(* PLC project liner_cyclic.project, CODESYS CODESYS V3.5 SP17 Patch 3 *)
(* stored: creationDateTime 1970-01-01T00:00:00, modificationDateTime 1970-01-01T00:00:00 *)

PROGRAM SafetyChain
  VAR
    BLINK_0 : BLINK;
    bHomePosition : BOOL;
    R_TRIG_0 : R_TRIG;
    UP : BOOL;
    DOWN : BOOL;
    R_TRIG_2 : R_TRIG;
    tTimeLow : TIME := TIME#1s0ms;
    tTimeHigh : TIME := TIME#2s0ms;
    GREEN : BOOL;
    BLINK_1 : BLINK;
    GREEN_BLINK : BOOL;
    out_blink : BOOL;
    R_TRIG_8 : R_TRIG;
    TON_0 : TON;
    R_TRIG_1 : R_TRIG;
    RED : BOOL;
  END_VAR
  VAR  (* added by the conversion: wires and edge detectors of the diagram *)
    _GE47_ENO : BOOL;
    _GE47_OUT : BOOL;
    _LE51_ENO : BOOL;
    _LE51_OUT : BOOL;
    _GE55_ENO : BOOL;
    _GE55_OUT : BOOL;
  END_VAR

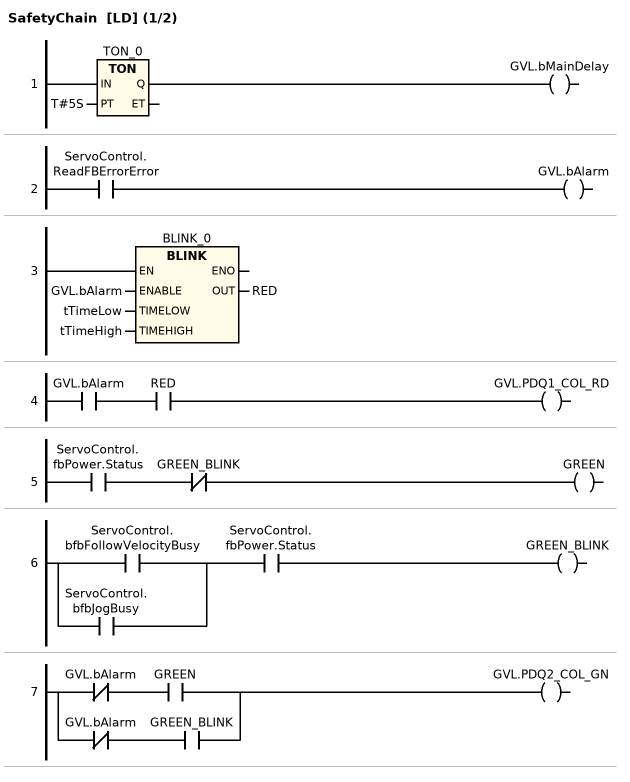
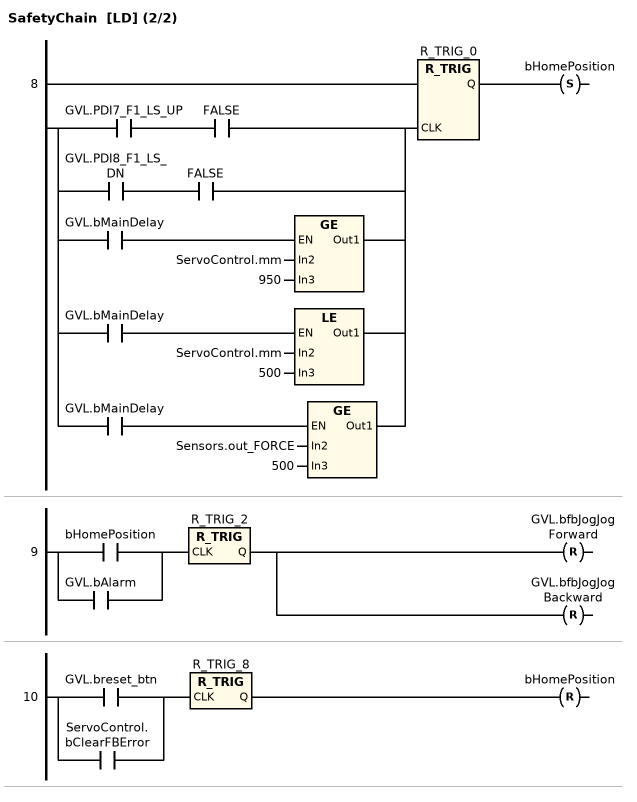
(* LD diagram, written out as Structured Text *)

TON_0(IN := TRUE, PT := T#5S);
GVL.bMainDelay := TON_0.Q;

GVL.bAlarm := ServoControl.ReadFBErrorError;

BLINK_0(ENABLE := GVL.bAlarm, TIMELOW := tTimeLow, TIMEHIGH := tTimeHigh, OUT => RED);

GVL.PDQ1_COL_RD := GVL.bAlarm AND RED;

GREEN := ServoControl.fbPower.Status AND NOT GREEN_BLINK;

GREEN_BLINK := (ServoControl.bfbFollowVelocityBusy OR ServoControl.bfbJogBusy) AND ServoControl.fbPower.Status;

GVL.PDQ2_COL_GN := NOT GVL.bAlarm AND (GREEN OR GREEN_BLINK);
(* 900мм - крайнее нижнее положение, 120 - крайнее верхнее положение *)

_GE47_OUT := GE(EN := GVL.bMainDelay, IN1 := ServoControl.mm, IN2 := 950, ENO => _GE47_ENO);
_LE51_OUT := LE(EN := GVL.bMainDelay, IN1 := ServoControl.mm, IN2 := 500, ENO => _LE51_ENO);
_GE55_OUT := GE(EN := GVL.bMainDelay, IN1 := Sensors.out_FORCE, IN2 := 500, ENO => _GE55_ENO);
R_TRIG_0(CLK := GVL.PDI7_F1_LS_UP AND FALSE OR GVL.PDI8_F1_LS_DN AND FALSE OR _GE47_OUT OR _LE51_OUT OR _GE55_OUT);
IF R_TRIG_0.Q THEN bHomePosition := TRUE; END_IF;
(* Отключаем JOG *)

R_TRIG_2(CLK := bHomePosition OR GVL.bAlarm);
IF R_TRIG_2.Q THEN GVL.bfbJogJogForward := FALSE; END_IF;
IF R_TRIG_2.Q THEN GVL.bfbJogJogBackward := FALSE; END_IF;
(* Принимаю за среднее положение значение от 499 до 501. Возврат в среднее положение при любых аварийных отклонениях. *)

R_TRIG_8(CLK := GVL.breset_btn OR ServoControl.bClearFBError);
IF R_TRIG_8.Q THEN bHomePosition := FALSE; END_IF;
END_PROGRAM
